Staubli VAL3: getFrameId.pgx

public program getFrameId(num& x_nFrame)
begin
end
